INTERFACE I_BoolValue EXTENDS __SYSTEM.IQueryInterface

{attribute 'monitoring' := 'call'}
PROPERTY Value : BOOL
GET
END_GET
END_PROPERTY

END_INTERFACE

(* stored: Version 1.1.0.1
   Itf I_BoolValue: Id {01d29d36-ba7c-4092-b1f5-74f7b21e0ae2}
   Property Value: Id {87675c9a-aa39-47a0-9993-c0c6c1a66444}
   Get Get: Id {47cd0bb6-72a2-4984-b13f-95db0f6a6103} *)
